PROGRAM MAIN
VAR
END_VAR

END_PROGRAM

(* stored: Version 1.1.0.1
   POU MAIN: Id {18f8347d-3537-4d3a-8104-11e436b81ca9} *)
